(* PLC project Unnamed, Unknown Unnamed 1 *)
(* stored: creationDateTime 2022-08-29T07:34:11, modificationDateTime 2022-09-01 14:53:16 *)

FUNCTION_BLOCK DEBOUNCE
  VAR_INPUT
    IN : BOOL;
    DB_TIME : TIME :=  T#2s;
  END_VAR
  VAR_OUTPUT
    OUT : BOOL;
    ET_OFF : TIME;
  END_VAR
  VAR
    DB_ON : TON;
    DB_OFF : TON;
    DB_FF : SR;
  END_VAR
  VAR  (* added by the conversion: wires and edge detectors of the diagram *)
    _NOT15_OUT : BOOL;
  END_VAR

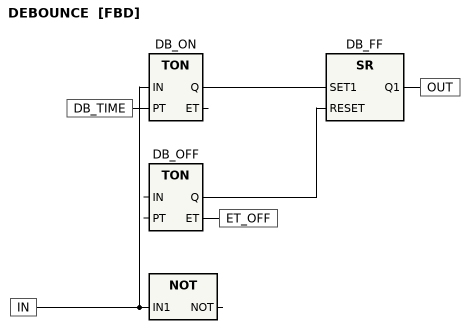
(* FBD diagram, written out as Structured Text *)
DB_ON(IN := IN, PT := DB_TIME);
DB_OFF();
DB_FF(SET1 := DB_ON.Q, RESET := DB_OFF.Q);
OUT := DB_FF.Q1;
ET_OFF := DB_OFF.ET;
_NOT15_OUT := NOT IN;
END_FUNCTION_BLOCK

(* LD *)
FUNCTION_BLOCK functionBlock0
  VAR
    A : BOOL;
    B : BOOL;
    C : BOOL;
  END_VAR

            LD    A
ANDN  B
ST    C













          
END_FUNCTION_BLOCK

FUNCTION_BLOCK functionBlock1
  VAR
    A : BOOL;
    B : BOOL;
    C : BOOL;
  END_VAR

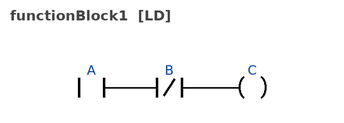
(* LD diagram, written out as Structured Text *)
C := A AND NOT B;
END_FUNCTION_BLOCK

FUNCTION_BLOCK functionBlock2
  VAR
    A : BOOL;
    B : BOOL;
    C : BOOL;
  END_VAR

            C := A AND NOT B;








          
END_FUNCTION_BLOCK

FUNCTION_BLOCK functionBlock3
  VAR
    A : BOOL;
    B : BOOL;
    C : BOOL;
  END_VAR

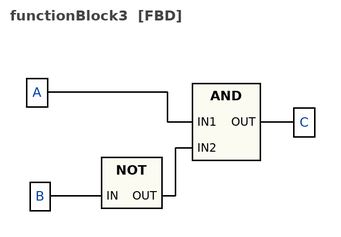
(* FBD diagram, written out as Structured Text *)
C := A AND NOT B;
END_FUNCTION_BLOCK

FUNCTION_BLOCK functionBlock4
  VAR
    A : BOOL;
    B : BOOL;
    C : BOOL;
  END_VAR

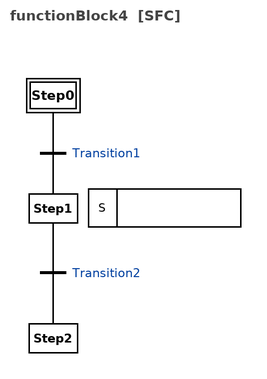
INITIAL_STEP Step0:
END_STEP
TRANSITION FROM Step0 TO Step1
  := Transition1;
END_TRANSITION
STEP Step1:
END_STEP
TRANSITION FROM Step1 TO Step2
  := Transition2;
END_TRANSITION
STEP Step2:
END_STEP
END_FUNCTION_BLOCK

CONFIGURATION config
  RESOURCE resource1 ON PLC
  END_RESOURCE
END_CONFIGURATION
